(* PLC project safeApp1, BrAutomation SafeDESIGNER  5.16.0.0 *)
(* stored: companyURL http://www.br-automation.com, creationDateTime Wed Mar 16 13:38:40 2022 *)

PROGRAM Main
  VAR  (* added by the conversion: wires and edge detectors of the diagram *)
    _AND_S12_OUT : ANY;
    _AND_S8_OUT : ANY;
    _AND_S29_OUT : ANY;
    _AND_S37_OUT : ANY;
  END_VAR

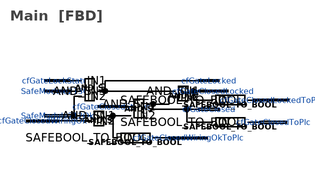
(* FBD diagram, written out as Structured Text *)
_AND_S12_OUT := AND_S(cfGateLockStatus, SafeModule213Ok, SafeModule212Ok);
cfGateLocked := _AND_S12_OUT;
_AND_S8_OUT := AND_S(SafeModule212Ok, cfGateClosedWiringOk);
_AND_S29_OUT := AND_S(cfGateClosedStatus, _AND_S8_OUT);
_AND_S37_OUT := AND_S(_AND_S12_OUT, _AND_S29_OUT);
cfGateClosedLocked := _AND_S37_OUT;
cfGateClosed := _AND_S29_OUT;
cfGateClosedLockedToPlc := SAFEBOOL_TO_BOOL(_AND_S37_OUT);
cfGateClosedToPlc := SAFEBOOL_TO_BOOL(_AND_S29_OUT);
cfGateClosedWiringOkToPlc := SAFEBOOL_TO_BOOL(_AND_S8_OUT);
END_PROGRAM
